// TIA Portal V19 export
TYPE "TAx_STATUSWORD"
// stored: Access Published
   STRUCT
      Enable : Bool;
      Error : Bool;
      RestartActive : Bool;
      OnlineStartValuesChanged : Bool;   // 0: Restart variable not changed; 1: Restart variable changed, TObject needs to be restarted
      ControlPanelActive : Bool;
      HomingDone : Bool;
      Done : Bool;   // 0: Last Job not done; 1: Last Job Done
      Standstill : Bool;
      PositioningCommand : Bool;
      JogCommand : Bool;
      VelocityCommand : Bool;
      HomingCommand : Bool;
      CostantVelocity : Bool;   // 1: Target speed reached;
      Accelerating : Bool;
      Decelerating : Bool;
      SW_NegativeLimitSwitch : Bool;   // 1: Limit switch engaged
      SW_PositiveLimitSwitch : Bool;   // 1: Limit switch engaged
      HW_NegativeLimitSwitch : Bool;   // 1: Limit switch engaged
      HW_PositiveLimitSwitch : Bool;   // 1: Limit switch engaged
      Bit_19 : Bool;   // Reserved
      Bit_20 : Bool;   // Reserved
      Synchronizing : Bool;   // Reserved - 1: Start synchronization with master
      Synchronous : Bool;   // Reserved - 1: Synchronized motion with master
      SuperimposedMotionCommand : Bool;
      PhasingCommand : Bool;
      AxisSimulation : Bool;   // 1: Simulation is active
      TorqueLimitingCommand : Bool;
      InLimitation : Bool;   // 1: Torque limiting is active
      NonPositionControlled : Bool;
      KinematicsMotionCommand : Bool;   // Reserve bit 5
      InClamping : Bool;
      MotionInCommand : Bool;   // Reserved
   END_STRUCT;
END_TYPE
